TYPE St_DataHisto_Epoch :
STRUCT
	Timestamp		: ULINT;
	ParentId		: DINT;
	Value			: LREAL;
END_STRUCT
END_TYPE

(* stored: Version 1.1.0.1, ProductVersion 3.1.4024.6
   DUT St_DataHisto_Epoch: Id {4bb549d8-1eb2-48c1-9098-6c4fc18ff80f} *)
